// TwinCAT 3 PLC project VAC_PLC
// ProgramVersion: 3.1.4020.5
// libraries:
//   L2SI Vacuum Library, * (SLAC)
//   Tc2_Standard, * (Beckhoff Automation GmbH)
//   Tc2_System, * (Beckhoff Automation GmbH)
//   Tc3_Module, * (Beckhoff Automation GmbH)
// project tree:
//   GVLs/ GVL_Devices.TcGVL
//   / PlcTask.TcTTO
//   POUs/ MAIN.TcPOU, POU_Example.TcPOU
// real-time tasks:
//   TASK PlcTask: cycle T#10ms, priority 20, ADS port 350

CONFIGURATION VAC_PLC
    RESOURCE PLC ON TwinCAT3
        TASK PlcTask(INTERVAL := T#10ms, PRIORITY := 20);
        PROGRAM MAIN WITH PlcTask : MAIN;
    END_RESOURCE
END_CONFIGURATION

// ---- GVLs/GVL_Devices.TcGVL

VAR_GLOBAL

	{attribute 'pytmc' := '
    pv: FEE:GPI:01
	'}
	FEE_GPI_01 : FB_MKS275;
	{attribute 'pytmc' := '
    pv: FEE:GCC:01
	'}
	FEE_GCC_01: FB_MKS500;	

	{attribute 'pytmc' := '
    pv: FEE:VGC:01
	'}
	FEE_VGC_01: FB_VGC;	
	
	
	{attribute 'pytmc' := '
    pv: FEE:GPI:02
	'}
	FEE_GPI_02 : FB_MKS275;
	{attribute 'pytmc' := '
    pv: FEE:GCC:02
	'}
	FEE_GCC_02: FB_MKS500;	
	
	{attribute 'pytmc' := '
    pv: FEE:PIP:01
	'}
	FEE_PIP_01: FB_PIP_Gamma;	

END_VAR

// ---- POUs/MAIN.TcPOU

PROGRAM MAIN
VAR

END_VAR

POU_Example();

END_PROGRAM

// ---- POUs/POU_Example.TcPOU
PROGRAM POU_Example
VAR
END_VAR

(* Here we call all the function block that have been declared in GVL_Devices*)


//Pirani Gauges
FEE_GPI_01();
FEE_GPI_02(PG=>);
// Ion Gauges
FEE_GCC_01(PG:= FEE_GPI_01.PG);
FEE_GCC_02(PG:= FEE_GPI_02.PG, IG=>);

//Isolation Valves
FEE_VGC_01(i_stUSG := FEE_GCC_01.IG, i_stDSG := FEE_GCC_02.IG, i_xDis_DPIlk:=TRUE, i_xEPS_OK:= TRUE, i_xPMPS_OK :=TRUE);

//Ion Pumps

END_PROGRAM
